FUNCTION_BLOCK FB_SecondObject
VAR_INPUT
END_VAR
VAR_OUTPUT
END_VAR
VAR
	_parentObject : ITF_Object;
	hResult : INT;
END_VAR

METHOD AttemptCast : BOOL
VAR_INPUT
END_VAR
VAR
	itfChild : ITF_ObjectExt;
END_VAR
IF __QUERYINTERFACE(_parentObject,itfChild) THEN
	hResult := itfChild.AddSomeValues(2,2);
	AttemptCast := TRUE;
END_IF
END_METHOD

PROPERTY ParentObject : ITF_Object
GET
ParentObject := _parentObject;
END_GET
SET
_parentObject := ParentObject;
END_SET
END_PROPERTY

END_FUNCTION_BLOCK

(* stored: Version 1.1.0.1, ProductVersion 3.1.4024.11
   POU FB_SecondObject: Id {fbd3061f-5804-4489-9875-37b80a2f97b3}, SpecialFunc None
   Method AttemptCast: Id {df8cd038-645c-4135-9171-9ef57d6861a3}
   Property ParentObject: Id {c7e52004-28a9-4ee7-9d15-00f540ed35e3}
   Get Get: Id {13707b24-db25-4573-9c5e-7d14fa01fecd}
   Set Set: Id {2feaec1f-fbca-4cfc-80ad-b60d68131550} *)
